// TwinCAT 3 PLC project Reservoir
// ProgramVersion: 3.1.4024.0
// libraries:
//   Tc2_MC2, * (Beckhoff Automation GmbH)
//   Tc2_NC, * (Beckhoff Automation GmbH)
//   Tc2_Standard, * (Beckhoff Automation GmbH)
//   Tc2_System, * (Beckhoff Automation GmbH)
//   Tc3_Module, * (Beckhoff Automation GmbH)
//   VisuDialogs, * (System)
// project tree:
//   / GlobalTextList.TcGTLO, PlcTask.TcTTO, Visualization Manager.TcVMO (not stored)
//   POUs/ LevelControl.TcPOU, MAIN.TcPOU, Reservoir.TcPOU, Visualization.TcVIS
// real-time tasks:
//   TASK PlcTask: cycle T#10ms, priority 20, ADS port 350
// motion (NC):
//   TASK AxisReservoir SAF: cycle T#2ms, priority 4, ADS port 501
//   TASK AxisReservoir SVB: cycle T#10ms, priority 8, ADS port 511
//   AXIS Agitator (id 1)
//     OtherSettings: AllowMotionCmdToSlave=true
//     encoder EncType=1
//     drive DrvType=5
//       Analog: TorqueSetpointScale=10, ScaleFactorActTorque=0.1
//       TimeComp: TaskDelayCycles=1
//     controller CtrType=1
//       CtrPara: PriorControlFactor=1
//         Observer: BandWidth=20
//   AXIS Pump (id 2)
//     OtherSettings: AllowMotionCmdToSlave=true
//     encoder EncType=1
//     drive DrvType=5
//       Analog: TorqueSetpointScale=10, ScaleFactorActTorque=0.1
//       TimeComp: TaskDelayCycles=1
//     controller CtrType=1
//       CtrPara: PriorControlFactor=1
//         Observer: BandWidth=20
// variable links:
//   Reservoir/Reservoir Instance <-> AxisReservoir SAF/Axes/Agitator
//     PlcTask Inputs/Reservoir.fbLevelCtrl.Agitator.NcToPlc <-> Outputs/ToPlc
//     PlcTask Outputs/Reservoir.fbLevelCtrl.Agitator.PlcToNc <-> Inputs/FromPlc
//   Reservoir/Reservoir Instance <-> AxisReservoir SAF/Axes/Pump
//     PlcTask Inputs/Reservoir.fbLevelCtrl.Pump.NcToPlc <-> Outputs/ToPlc
//     PlcTask Outputs/Reservoir.fbLevelCtrl.Pump.PlcToNc <-> Inputs/FromPlc

CONFIGURATION Reservoir
    RESOURCE PLC ON TwinCAT3
        TASK PlcTask(INTERVAL := T#10ms, PRIORITY := 20);
        PROGRAM MAIN WITH PlcTask : MAIN;
    END_RESOURCE
END_CONFIGURATION

// ---- POUs/MAIN.TcPOU
PROGRAM MAIN
VAR
END_VAR

Reservoir();

END_PROGRAM

// ---- POUs/Reservoir.TcPOU
PROGRAM Reservoir
VAR
	fbLevelCtrl : LevelControl;
	bLowLevelAlarm : BOOL;
	bHighLevelAlarm : BOOL;
	
	bResetButton : BOOL;
	bStartButton : BOOL;
	bStopButton : BOOL;
	
	bPumpLight : BOOL;
	bAgitatorLight : BOOL;
	bSolenoidALight : BOOL;
	bSolenoidBLight : BOOL;
	
	rSensorInput : REAL;
	
	rPumpOutput : LREAL;
	rAgitatorOutput : LREAL;
END_VAR

bLowLevelAlarm := fbLevelCtrl.bLowLevel;
bHighLevelAlarm := fbLevelCtrl.bHighLevel;

fbLevelCtrl.bStart := bStartButton;
fbLevelCtrl.bStop := bStopButton;
fbLevelCtrl.bReset := bResetButton;

bPumpLight := fbLevelCtrl.bPump;
bAgitatorLight := fbLevelCtrl.bAgitator;
bSolenoidALight := fbLevelCtrl.bSolenoidA;
bSolenoidBLight := fbLevelCtrl.bSolenoidB;

fbLevelCtrl.rWaterLevel := rSensorInput;

rPumpOutput := fbLevelCtrl.rPumpPos;
rAgitatorOutput := fbLevelCtrl.rAgitatorPos;


fbLevelCtrl();

END_PROGRAM

// ---- POUs/LevelControl.TcPOU
FUNCTION_BLOCK LevelControl
VAR_INPUT
	bStart : BOOL;
	bStop : BOOL;
	bReset : BOOL;
	
	rWaterLevel : REAL;
END_VAR
VAR_OUTPUT
	bHighLevel : BOOL;
	bLowLevel : BOOL;
	
	bSolenoidA : BOOL;
	bSolenoidB : BOOL;
	
	bPump : BOOL;
	bAgitator : BOOL;
	
	rPumpPos : LREAL;
	rAgitatorPos : LREAL;
END_VAR
VAR
	iState : UDINT;
	bInitialActivate : BOOL;
	
	fbInitial : R_TRIG;
	
	Agitator : AXIS_REF;
	Pump : AXIS_REF;
	JogAgitator : MC_Jog;
	JogPump : MC_Jog;
	PowerAgitator : MC_Power;
	PowerPump : MC_Power;
END_VAR

bInitialActivate := TRUE; 
fbInitial(CLK := TRUE);
IF fbInitial.Q THEN
	rWaterLevel := 0.0; //sets the starting point for level to 0
END_IF
IF bStart THEN
	JogAgitator(Axis := Agitator,JogForward := TRUE);
END_IF
IF bStop THEN
	JogAgitator(Axis := Agitator,JogForward := FALSE);
END_IF

IF JogPump.Active THEN
	bPump := TRUE;
ELSIF NOT JogPump.Active THEN
	bPump := FALSE;	
END_IF

IF JogAgitator.Active THEN
	bAgitator := TRUE;
ELSIF NOT JogAgitator.Active THEN
	bAgitator := FALSE;	
END_IF

CASE iState OF
	0:
		IF PowerAgitator.Status AND PowerPump.Status THEN
			iState := 10;
		END_IF
	5: //if agitator is turned off reset
		JogPump(Axis := Pump,JogForward := FALSE);
		bSolenoidA := FALSE;
		bSolenoidB := FALSE;
		iState := 0;	
	10://check the water level
		IF JogAgitator.Active THEN
			IF rWaterLevel >= 9.5 AND rWaterLevel < 24.5 THEN
				iState := 20;
			ELSIF rWaterLevel >= 24.5	AND rWaterLevel < 89.5 THEN
				iState := 30;
			ELSIF rWaterLevel < 9.5 AND rWaterLevel > 0.0 THEN
				iState := 40;
			ELSIF rWaterLevel >= 89.5 THEN
				iState := 50;
			END_IF
		END_IF
	20: //fill the reservoir
		IF JogAgitator.Active THEN
			bSolenoidA := TRUE;
			bSolenoidB := TRUE;
			JogPump(Axis := Pump,JogForward := FALSE);
			bHighLevel := FALSE;
			bLowLevel := FALSE;
			iState := 0;
		ELSE
			iState := 5;	
		END_IF
	30: //empty the reservoir
		IF JogAgitator.Active THEN
			JogPump(Axis := Pump,JogForward := TRUE);
			bSolenoidA := FALSE;
			bSolenoidB := FALSE;
			bHighLevel := FALSE;
			bLowLevel := FALSE;
			iState := 0;
		ELSE
			iState := 5;	
		END_IF
	40: //crtitically low level
		IF JogAgitator.Active THEN
			bSolenoidA := FALSE;
			bSolenoidB := FALSE;
			JogPump(Axis := Pump,JogForward := FALSE);
			bHighLevel := FALSE;
			bLowLevel := TRUE;
			IF bReset  THEN
				iState := 100;
			END_IF
		ELSE
			iState := 5;	
		END_IF
	50: //critically high level	
		IF JogAgitator.Active THEN
			bSolenoidA := FALSE;
			bSolenoidB := FALSE;
			JogPump(Axis := Pump,JogForward := FALSE);
			bHighLevel := TRUE;
			bLowLevel := FALSE;
			IF bReset  THEN
				iState := 100;
			END_IF
		ELSE
			iState := 5;	
		END_IF
	100://reset
		bLowLevel := FALSE;
		bHighLevel := FALSE;
		iState := 0;
			 		
END_CASE

PowerAgitator(Axis := Agitator,Enable := TRUE,Enable_Positive := TRUE,Enable_Negative := TRUE);
PowerPump(Axis := Pump,Enable := TRUE,Enable_Positive := TRUE,Enable_Negative := TRUE);

JogAgitator(Axis := Agitator);
JogPump(Axis := Pump);

rPumpPos := Pump.NcToPlc.ActPos;
rAgitatorPos := Agitator.NcToPlc.ActPos;

END_FUNCTION_BLOCK

// ---- GlobalTextList.TcGTLO
TEXTLIST GlobalTextList
  753 = '%f'
  197 = '%f Sensor Input'
  58 = '%i'
  954 = '%lr'
  507 = '%r'
  949 = '%r  Sensor Input'
  504 = '%r Sensor Input'
  171 = 'Agitator'
  975 = 'High Level'
  391 = 'Low Level'
  816 = 'PUMP'
  503 = 'Reset'
  966 = 'Sensor Input'
  703 = 'Solenoid A'
  189 = 'Solenoid B'
  46 = 'Start'
  769 = 'Stop'
END_TEXTLIST

// ---- POUs/Visualization.TcVIS
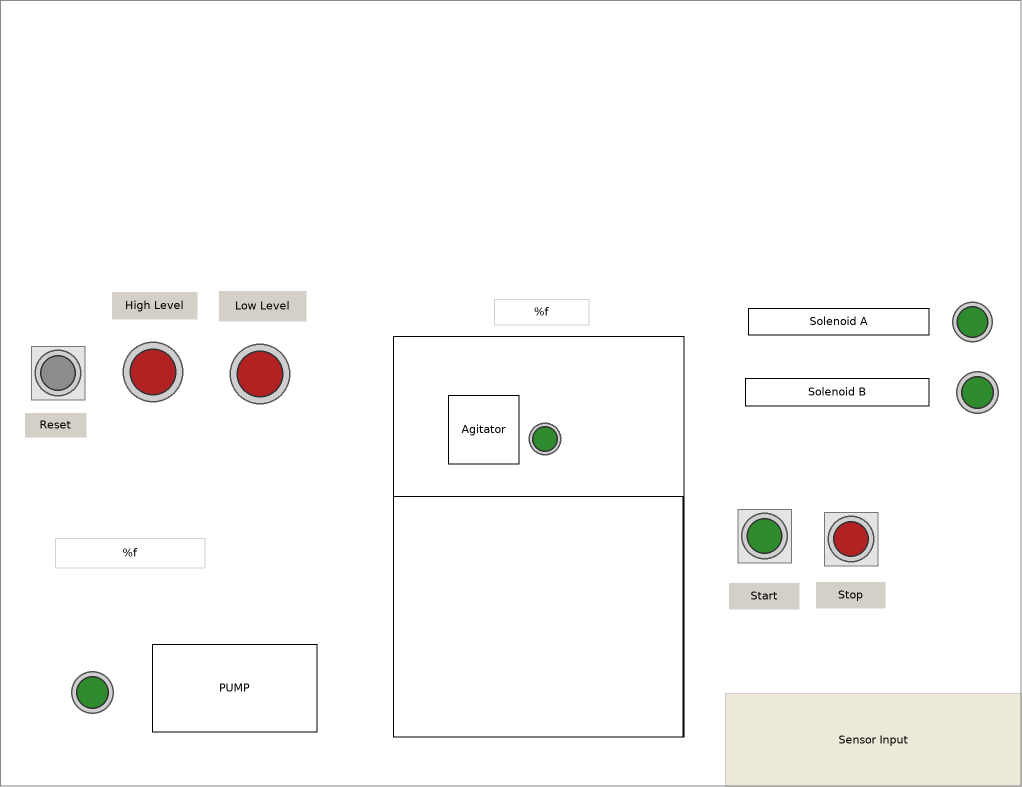
VISUALIZATION Visualization  // 1022x787
    Rectangle (393,336 291x401)
    Rectangle (393,496 290x241)
    Lamp1 (118,337 70x70), variable: Reservoir.bHighLevelAlarm, style: Lamp-Lamp1-Red
    Lamp1 (225,339 70x70), variable: Reservoir.bLowLevelAlarm, style: Lamp-Lamp1-Red
    Lamp1 (949,297 47x50), variable: Reservoir.bSolenoidALight, style: Lamp-Lamp1-Green
    Lamp1 (949,368 57x49), variable: Reservoir.bSolenoidBLight, style: Lamp-Lamp1-Green
    Lamp1 (526,413 38x52), variable: Reservoir.bAgitatorLight, style: Lamp-Lamp1-Green
    Lamp1 (68,665 49x55), variable: Reservoir.bPumpLight, style: Lamp-Lamp1-Green
    Rectangle (152,644 165x88), "PUMP"
    Rectangle (748,308 181x27), "Solenoid A"
    Rectangle (745,378 184x28), "Solenoid B"
    Rectangle (448,395 71x69), "Agitator"
    PushSwitch (31,345 54x56), variable: Reservoir.bResetButton, behaviour: TAP, style: Switch-PushSwitch-Gray
    PushSwitch (824,508 54x62), variable: Reservoir.bStopButton, behaviour: TAP, style: Switch-PushSwitch-Red
    PushSwitch (737,509 55x54), variable: Reservoir.bStartButton, behaviour: TAP, style: Switch-PushSwitch-Green
    Textfield (729,583 70x26), "Start"
    Textfield (816,582 69x26), "Stop"
    Textfield (25,413 61x24), "Reset"
    Textfield (112,292 85x27), "High Level"
    Textfield (219,291 87x30), "Low Level"
    Textfield (725,693 297x94), "Sensor Input", text variable: Reservoir.rSensorInput
        OnMouseDown: write the text variable via Default
    Textfield (55,538 150x30), "%f", text variable: Reservoir.rPumpOutput
    Textfield (494,299 95x26), "%f", text variable: Reservoir.rAgitatorOutput
END_VISUALIZATION
